(* IEC 61131-3 sources: MyTestRepos/MyPlcProject, 2 files *)

(* ---- GlobalVariables.gvl ---- *)
VAR_GLOBAL

END_VAR

(* ---- PLC_PRG.st ---- *)
PROGRAM PLC_PRG
VAR
	myVar : INT;
END_VAR

myVar := 46;
END_PROGRAM

ACTIONS

END_ACTIONS
